// Mitsubishi GX Works2 project: PLC_Group_16   PLC: FX3G

// global labels: Global1
VAR_GLOBAL
  StartWorkingDay AT X010 : BOOL;
  In_Flour AT D1101 : REAL;
  Flour_Stock AT D1111 : REAL;
  check AT M0 : BOOL;
  In_Yeast AT D1103 : REAL;
  In_Water AT D1105 : REAL;
  In_Oil AT D1107 : REAL;
  In_Spice AT D1109 : REAL;
  Yeast_Stock AT D1113 : REAL;
  Water_Stock AT D1115 : REAL;
  Oil_Stock AT D1117 : REAL;
  Spice_Stock AT D1119 : REAL;
  Emergency_Button AT X007 : BOOL;
  Emg_Stop AT X007 : BOOL;
END_VAR
VAR_GLOBAL CONSTANT
  ratio1 : REAL := 0.2;
  Ratio_Yeast : REAL := 0.2;
END_VAR
VAR_GLOBAL
  Check_Yeast AT D1121 : REAL;
END_VAR
VAR_GLOBAL CONSTANT
  Ratio_Water : REAL := 0.5;
  Ratio_Oil : REAL := 0.3;
  Ratio_Spice : REAL := 0.1;
END_VAR
VAR_GLOBAL
  Check_Water AT D1123 : REAL;
  Check_Oil AT D1125 : REAL;
  Check_Spice AT D1127 : REAL;
END_VAR
VAR_GLOBAL CONSTANT
  MIN_Flour : REAL := 100.0;
END_VAR
VAR_GLOBAL
  checkY AT M1 : BOOL;
  checkW AT M2 : BOOL;
  checkO AT M3 : BOOL;
  checkS AT M4 : BOOL;
  checkF AT M5 : BOOL;
  active_workday AT Y010 : BOOL;
  M_10 AT M10 : BOOL;
  Start_Lisha AT X001 : BOOL;
  TC_1 AT TC1 : BOOL;
  TS_1 AT TS1 : BOOL;
  Lisha_Light AT Y001 : BOOL;
END_VAR
VAR_GLOBAL CONSTANT
  cons30 : INT := 30;
END_VAR
VAR_GLOBAL
  Water_Mixer AT D1131 : REAL;
  Flour_Mixer AT D1129 : REAL;
  Oil_Mixer AT D1133 : REAL;
  Spice_Mixer AT D1135 : REAL;
  Yeast_Mixer AT D1137 : REAL;
  Flour_Hatpaja AT D1139 : REAL;
  Water_Hatpaja AT D1141 : REAL;
  Yeat_Hatpaja AT D1143 : REAL;
  Oil_Hatpaja AT D1145 : REAL;
  Spice_Hatpaja AT D1147 : REAL;
  Flour_Bake AT D1149 : REAL;
  Water_Bake AT D1151 : REAL;
  Yeast_Bake AT D1153 : REAL;
  Oil_Bake AT D1155 : REAL;
  Spice_Bake AT D1157 : REAL;
  Flour_Store AT D1159 : REAL;
  Water_Store AT D1161 : REAL;
  Yeast_Store AT D1163 : REAL;
  Oil_Store AT D1165 : REAL;
  Spice_Store AT D1167 : REAL;
END_VAR
VAR_GLOBAL CONSTANT
  FlourCONS : REAL := 100;
  YeastCONS : REAL := 20;
  WaterCONS : REAL := 50;
  OilCONS : REAL := 30;
  SpiceCONS : REAL := 10;
END_VAR
VAR_GLOBAL
  checkREGISTER AT D1199 : REAL;
  Flour_Mehal AT D1169 : REAL;
  Water_Mehal AT D1171 : REAL;
  Oil_Mehal AT D1173 : REAL;
  Spice_Mehal AT D1175 : REAL;
  Yeast_Mehal AT D1177 : REAL;
  M_MEHAL AT M12 : BOOL;
  Start_Mehal AT X002 : BOOL;
  CC_1 AT CC1 : BOOL;
END_VAR
VAR_GLOBAL CONSTANT
  cons2 : INT := 2;
END_VAR
VAR_GLOBAL
  Start_Hatpaja AT X011 : BOOL;
  CS_1 AT CS1 : BOOL;
  Hachana_Light AT Y005 : BOOL;
  M_15 AT M15 : BOOL;
  M_11 AT M11 : BOOL;
  TC_2 AT TC2 : BOOL;
  TS_2 AT TS2 : BOOL;
  Hatpaja_Light_1 AT Y002 : BOOL;
  TC_3 AT TC3 : BOOL;
  TS_3 AT TS3 : BOOL;
  Hatpaja_Light_2 AT Y003 : BOOL;
END_VAR
VAR_GLOBAL CONSTANT
  cons20 : INT := 20;
END_VAR
VAR_GLOBAL
  TC_4 AT TC4 : BOOL;
END_VAR
VAR_GLOBAL CONSTANT
  Timer_3Sec : INT := 30;
END_VAR
VAR_GLOBAL
  TS_5 AT TS5 : BOOL;
  M_14 AT M14 : BOOL;
  TS_4 AT TS4 : BOOL;
END_VAR
VAR_GLOBAL CONSTANT
  cons5 : INT := 5;
END_VAR
VAR_GLOBAL
  TC_6 AT TC6 : BOOL;
END_VAR
VAR_GLOBAL CONSTANT
  cons40 : INT := 40;
END_VAR
VAR_GLOBAL
  TS_6 AT TS6 : BOOL;
  Bake_Light AT Y004 : BOOL;
  Start_Test AT X003 : BOOL;
  Analog_Input2 AT D8281 : INT;
  Analog_Test AT D8201 : INT;
END_VAR
VAR_GLOBAL CONSTANT
  Analog_Max : INT := 2000;
  Analog_Min : INT := 400;
END_VAR
VAR_GLOBAL
  M_6 AT M6 : BOOL;
  M_7 AT M7 : BOOL;
  TC_7 AT TC7 : BOOL;
  TS_7 AT TS7 : BOOL;
  Store_Light AT Y006 : BOOL;
  CC_3 AT CC3 : BOOL;
  CS_3 AT CS3 : BOOL;
  M_8 AT M8 : BOOL;
  TC_8 AT TC8 : BOOL;
  TC_9 AT TC9 : BOOL;
  TS_9 AT TS9 : BOOL;
  TC_10 AT TC10 : BOOL;
  M_30 AT M30 : BOOL;
  M_31 AT M31 : BOOL;
  TS_10 AT TS10 : BOOL;
END_VAR
VAR_GLOBAL CONSTANT
  Materials : BOOL := TRUE;
  Empty : BOOL;
END_VAR
VAR_GLOBAL
  M_32 AT M32 : BOOL;
  M_33 AT M33 : BOOL;
  FinishWorkingDay AT M34 : BOOL;
  M_40 AT M40 : BOOL;
  M_41 AT M41 : BOOL;
  M_42 AT M42 : BOOL;
  M_43 AT M43 : BOOL;
  M_44 AT M44 : BOOL;
  M_45 AT M45 : BOOL;
  M_46 AT M46 : BOOL;
  M_47 AT M47 : BOOL;
  M_48 AT M48 : BOOL;
  M_49 AT M49 : BOOL;
  M_FinishRound AT M50 : BOOL;
END_VAR
VAR_GLOBAL CONSTANT
  const0 : REAL;
END_VAR
VAR_GLOBAL
  M_88 AT M88 : BOOL;
  M_89 AT M89 : BOOL;
  M_90 AT M90 : BOOL;
  M_91 AT M91 : BOOL;
  M_92 AT M92 : BOOL;
  Ipus AT M99 : BOOL;
END_VAR
VAR_GLOBAL CONSTANT
  cons0 : REAL;
END_VAR
VAR_GLOBAL
  M_111 AT M111 : BOOL;
END_VAR

// task Task_01 (event TRUE, interval 0, priority 31): POU_01

PROGRAM POU_01
(* structured ladder/FBD written out as ST: instructions are called as NAME(EN, inputs, outputs); _pN, _eN, _tN stand for wires *)
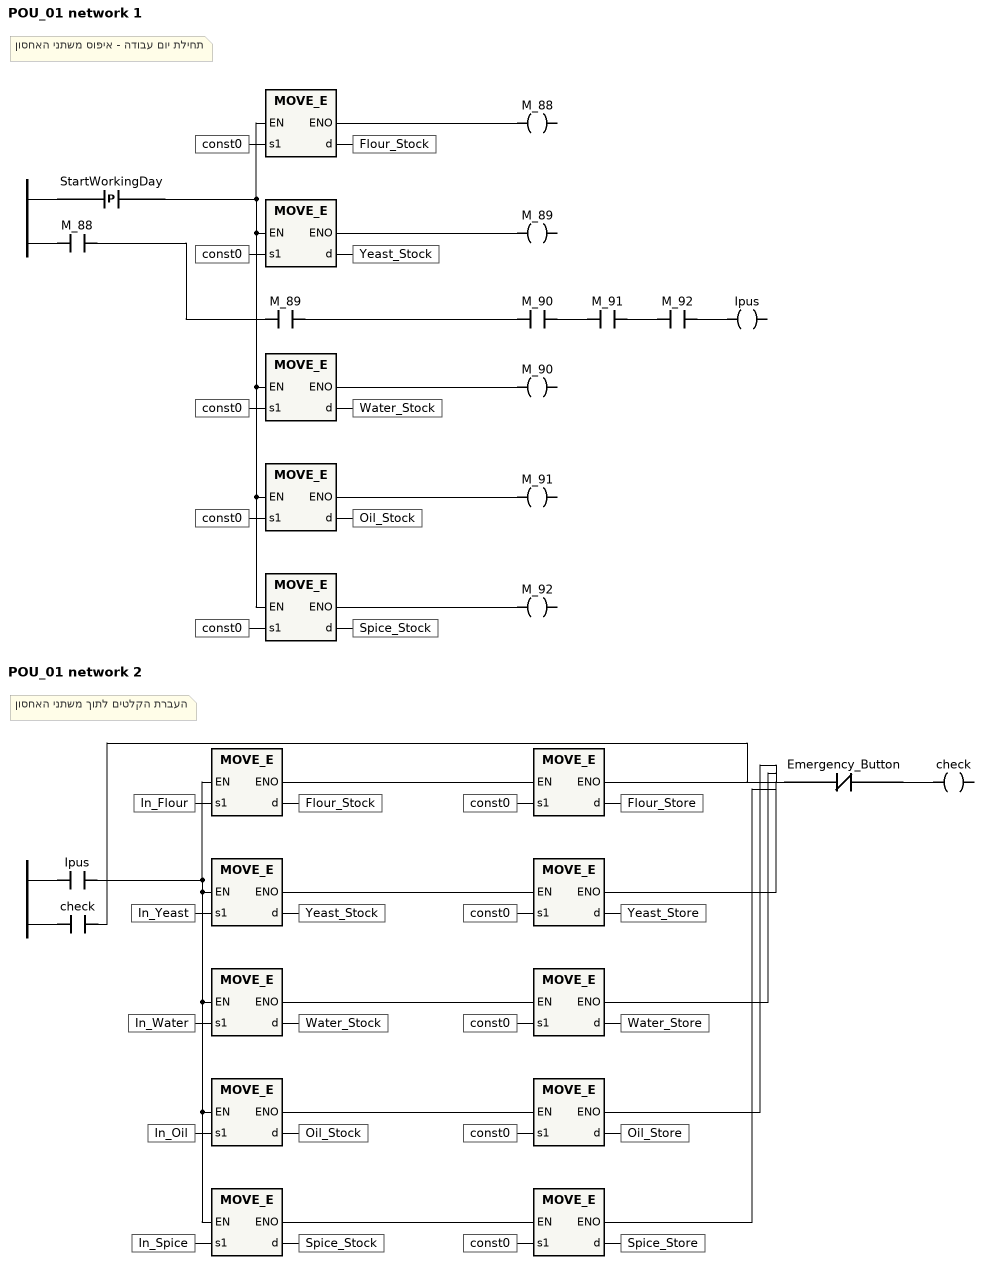
(* network 1 *)
(* תחילת יום עבודה - איפוס משתני האחסון *)
_p1 := LDP(TRUE, StartWorkingDay);
_e2 := MOVE_E(_p1, const0, Flour_Stock);
M_88 := _e2;
_e3 := MOVE_E(_p1, const0, Yeast_Stock);
M_89 := _e3;
_e4 := MOVE_E(_p1, const0, Water_Stock);
M_90 := _e4;
_e5 := MOVE_E(_p1, const0, Oil_Stock);
M_91 := _e5;
_e6 := MOVE_E(_p1, const0, Spice_Stock);
M_92 := _e6;
Ipus := M_88 AND M_89 AND M_90 AND M_91 AND M_92;
(* network 2 *)
(* העברת הקלטים לתוך משתני האחסון *)
_e1 := MOVE_E(Ipus, In_Flour, Flour_Stock);
_e2 := MOVE_E(_e1, const0, Flour_Store);
_e3 := MOVE_E(Ipus, In_Yeast, Yeast_Stock);
_e4 := MOVE_E(_e3, const0, Yeast_Store);
_e5 := MOVE_E(Ipus, In_Water, Water_Stock);
_e6 := MOVE_E(_e5, const0, Water_Store);
_e7 := MOVE_E(Ipus, In_Oil, Oil_Stock);
_e8 := MOVE_E(_e7, const0, Oil_Store);
_e9 := MOVE_E(Ipus, In_Spice, Spice_Stock);
_e10 := MOVE_E(_e9, const0, Spice_Store);
check := (_e2 OR _e4 OR _e6 OR _e8 OR _e10 OR check) AND NOT Emergency_Button;
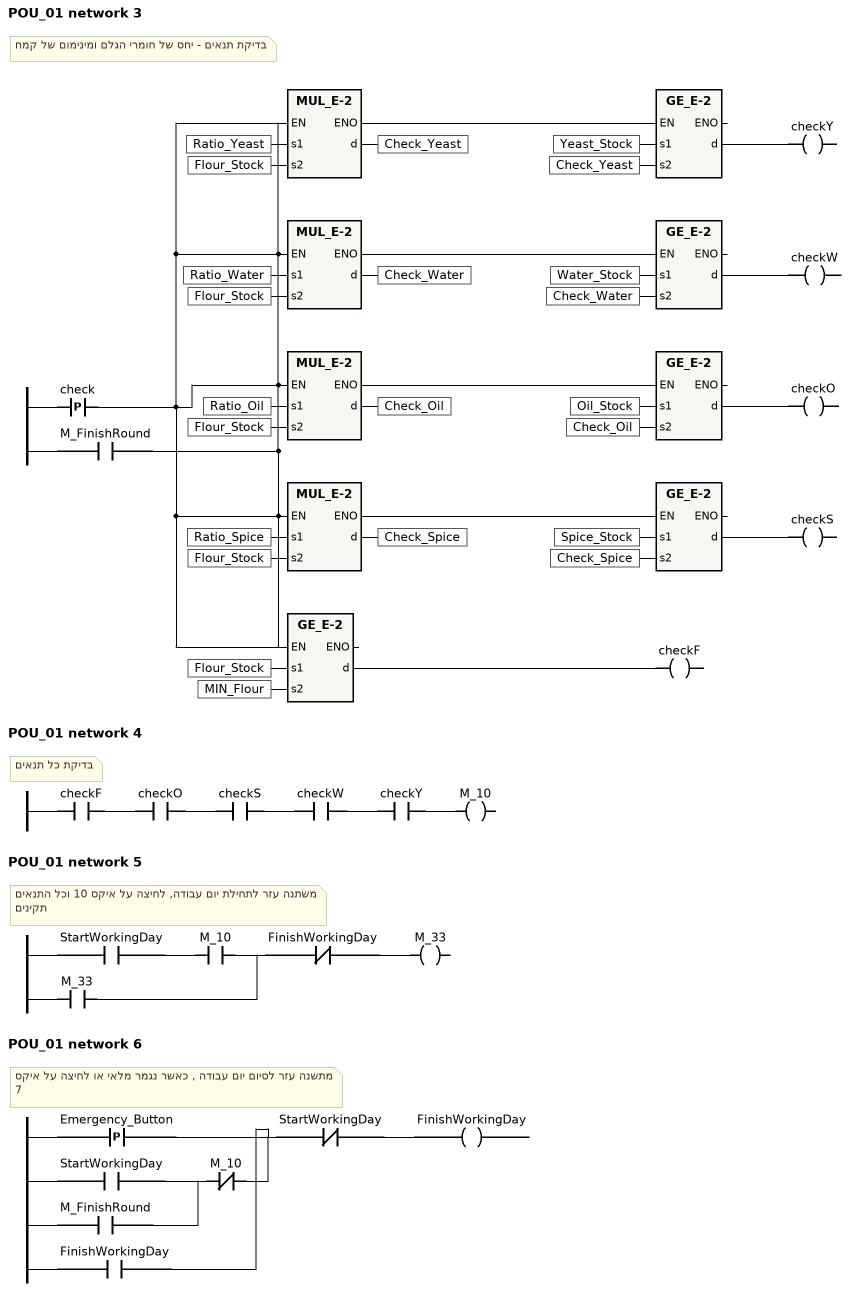
(* network 3 *)
(* בדיקת תנאים - יחס של חומרי הגלם ומינימום של קמח *)
_p1 := LDP(TRUE, check) OR M_FinishRound;
_e2 := MUL_E(_p1, Ratio_Yeast, Flour_Stock, Check_Yeast);
GE_E(_e2, Yeast_Stock, Check_Yeast, _t3);
checkY := _t3;
_e4 := MUL_E(_p1, Ratio_Water, Flour_Stock, Check_Water);
GE_E(_e4, Water_Stock, Check_Water, _t5);
checkW := _t5;
_e6 := MUL_E(_p1, Ratio_Oil, Flour_Stock, Check_Oil);
GE_E(_e6, Oil_Stock, Check_Oil, _t7);
checkO := _t7;
_e8 := MUL_E(_p1, Ratio_Spice, Flour_Stock, Check_Spice);
GE_E(_e8, Spice_Stock, Check_Spice, _t9);
checkS := _t9;
GE_E(_p1, Flour_Stock, MIN_Flour, _t10);
checkF := _t10;
(* network 4 *)
(* בדיקת כל תנאים *)
M_10 := checkF AND checkO AND checkS AND checkW AND checkY;
(* network 5 *)
(* משתנה עזר לתחילת יום עבודה, לחיצה על איקס 10 וכל התנאים תקינים *)
M_33 := ((StartWorkingDay AND M_10) OR M_33) AND NOT FinishWorkingDay;
(* network 6 *)
(* מתשנה עזר לסיום יום עבודה , כאשר נגמר מלאי או לחיצה על איקס 7 *)
FinishWorkingDay := (LDP(TRUE, Emergency_Button) OR ((StartWorkingDay OR M_FinishRound) AND NOT M_10) OR FinishWorkingDay) AND NOT StartWorkingDay;
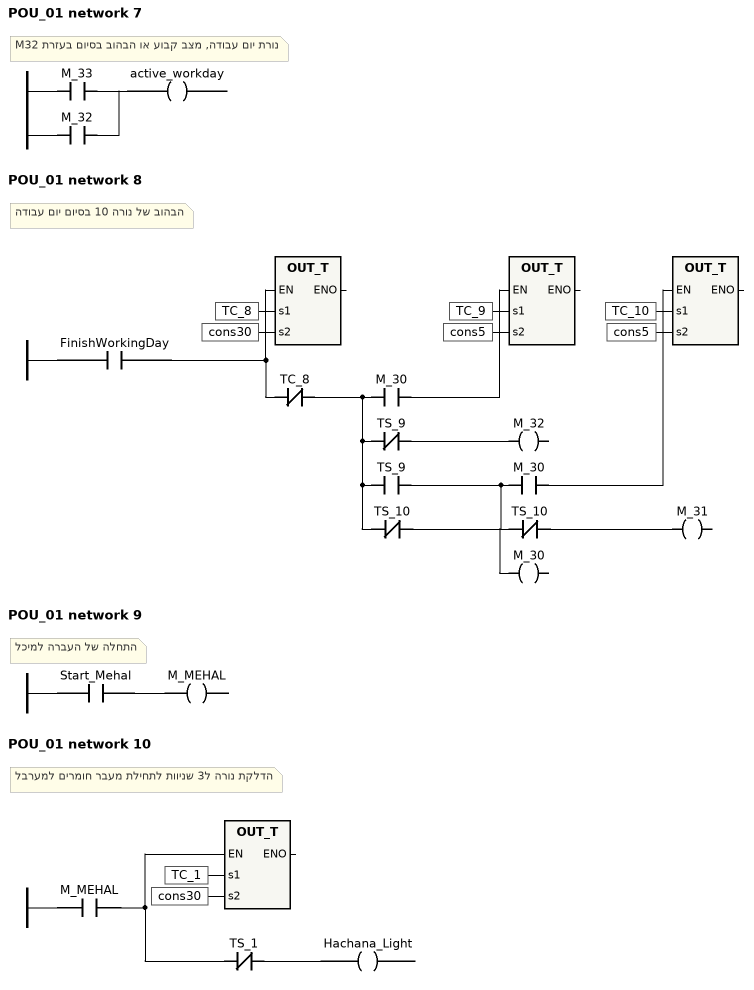
(* network 7 *)
(* נורת יום עבודה, מצב קבוע או הבהוב בסיום בעזרת M32 *)
active_workday := M_33 OR M_32;
(* network 8 *)
(* הבהוב של נורה 10 בסיום יום עבודה *)
OUT_T(FinishWorkingDay, TC_8, cons30);
_p1 := FinishWorkingDay AND NOT TC_8;
OUT_T(_p1 AND M_30, TC_9, cons5);
M_32 := _p1 AND NOT TS_9;
_p2 := _p1 AND TS_9;
OUT_T(_p2 AND M_30, TC_10, cons5);
M_31 := _p2 AND NOT TS_10;
M_30 := _p1 AND NOT TS_10;
(* network 9 *)
(* התחלה של העברה למיכל *)
M_MEHAL := Start_Mehal;
(* network 10 *)
(* הדלקת נורה ל3 שניוות לתחילת מעבר חומרים למערבל *)
OUT_T(M_MEHAL, TC_1, cons30);
Hachana_Light := M_MEHAL AND NOT TS_1;
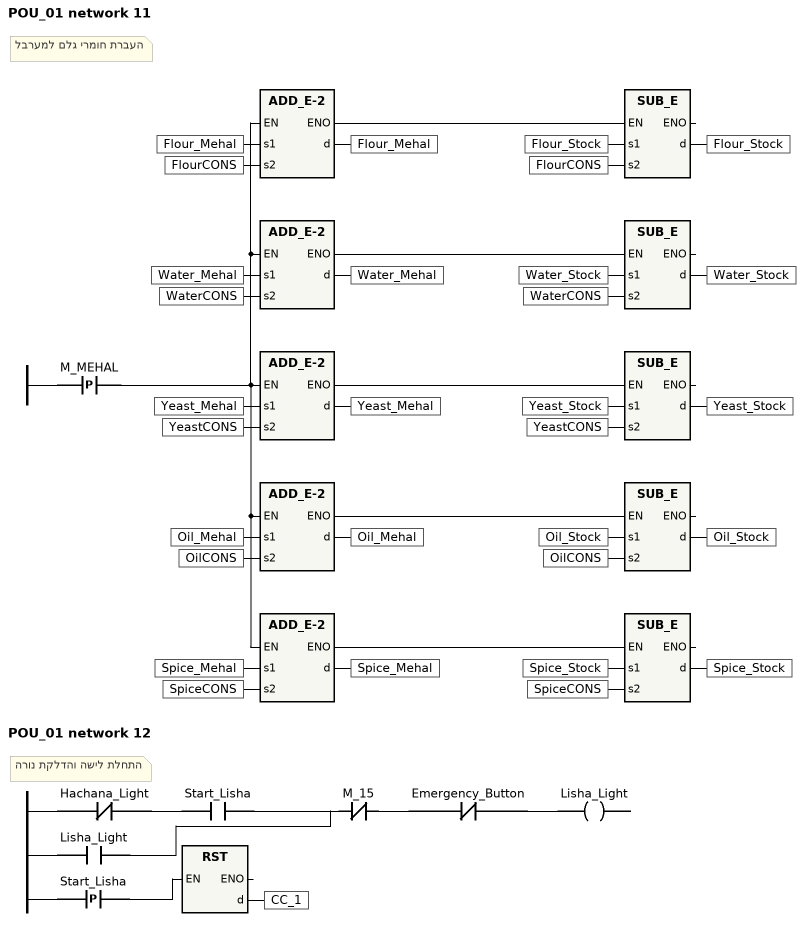
(* network 11 *)
(* העברת חומרי גלם למערבל *)
_p1 := LDP(TRUE, M_MEHAL);
_e2 := ADD_E(_p1, Flour_Mehal, FlourCONS, Flour_Mehal);
SUB_E(_e2, Flour_Stock, FlourCONS, Flour_Stock);
_e3 := ADD_E(_p1, Water_Mehal, WaterCONS, Water_Mehal);
SUB_E(_e3, Water_Stock, WaterCONS, Water_Stock);
_e4 := ADD_E(_p1, Yeast_Mehal, YeastCONS, Yeast_Mehal);
SUB_E(_e4, Yeast_Stock, YeastCONS, Yeast_Stock);
_e5 := ADD_E(_p1, Oil_Mehal, OilCONS, Oil_Mehal);
SUB_E(_e5, Oil_Stock, OilCONS, Oil_Stock);
_e6 := ADD_E(_p1, Spice_Mehal, SpiceCONS, Spice_Mehal);
SUB_E(_e6, Spice_Stock, SpiceCONS, Spice_Stock);
(* network 12 *)
(* התחלת לישה והדלקת נורה *)
Lisha_Light := (((NOT Hachana_Light AND Start_Lisha) OR Lisha_Light) AND NOT M_15) AND NOT Emergency_Button;
RST(LDP(TRUE, Start_Lisha), CC_1);
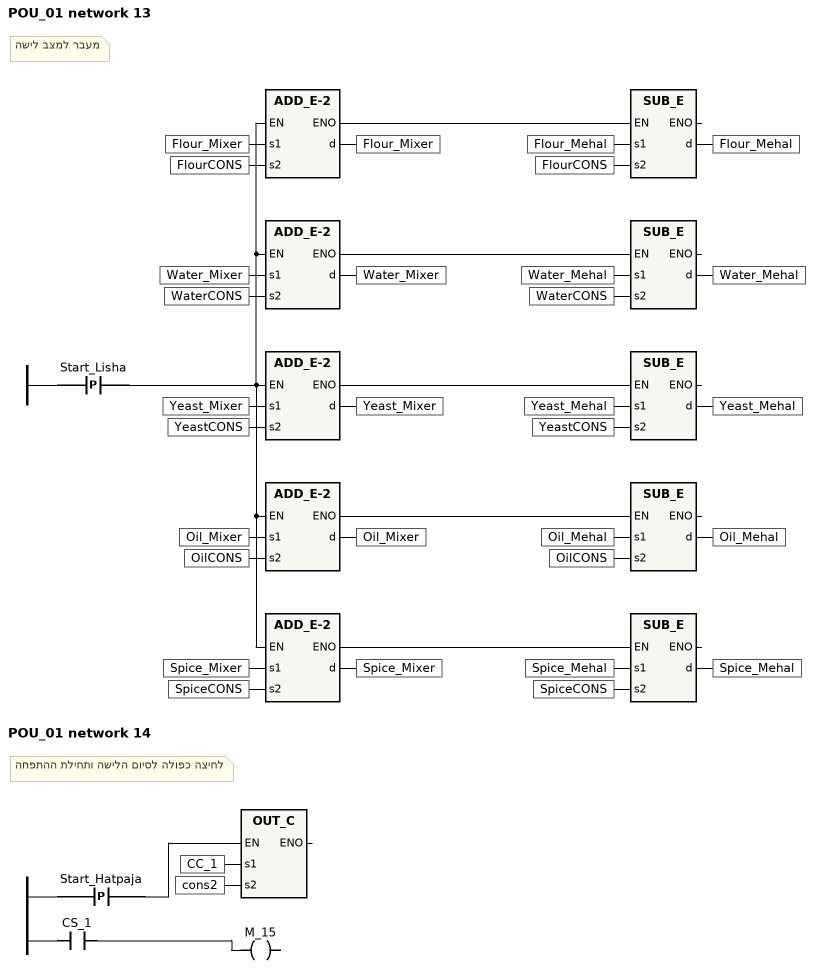
(* network 13 *)
(* מעבר למצב לישה *)
_p1 := LDP(TRUE, Start_Lisha);
_e2 := ADD_E(_p1, Flour_Mixer, FlourCONS, Flour_Mixer);
SUB_E(_e2, Flour_Mehal, FlourCONS, Flour_Mehal);
_e3 := ADD_E(_p1, Water_Mixer, WaterCONS, Water_Mixer);
SUB_E(_e3, Water_Mehal, WaterCONS, Water_Mehal);
_e4 := ADD_E(_p1, Yeast_Mixer, YeastCONS, Yeast_Mixer);
SUB_E(_e4, Yeast_Mehal, YeastCONS, Yeast_Mehal);
_e5 := ADD_E(_p1, Oil_Mixer, OilCONS, Oil_Mixer);
SUB_E(_e5, Oil_Mehal, OilCONS, Oil_Mehal);
_e6 := ADD_E(_p1, Spice_Mixer, SpiceCONS, Spice_Mixer);
SUB_E(_e6, Spice_Mehal, SpiceCONS, Spice_Mehal);
(* network 14 *)
(* לחיצה כפולה לסיום הלישה ותחילת ההתפחה *)
OUT_C(LDP(TRUE, Start_Hatpaja), CC_1, cons2);
M_15 := CS_1;
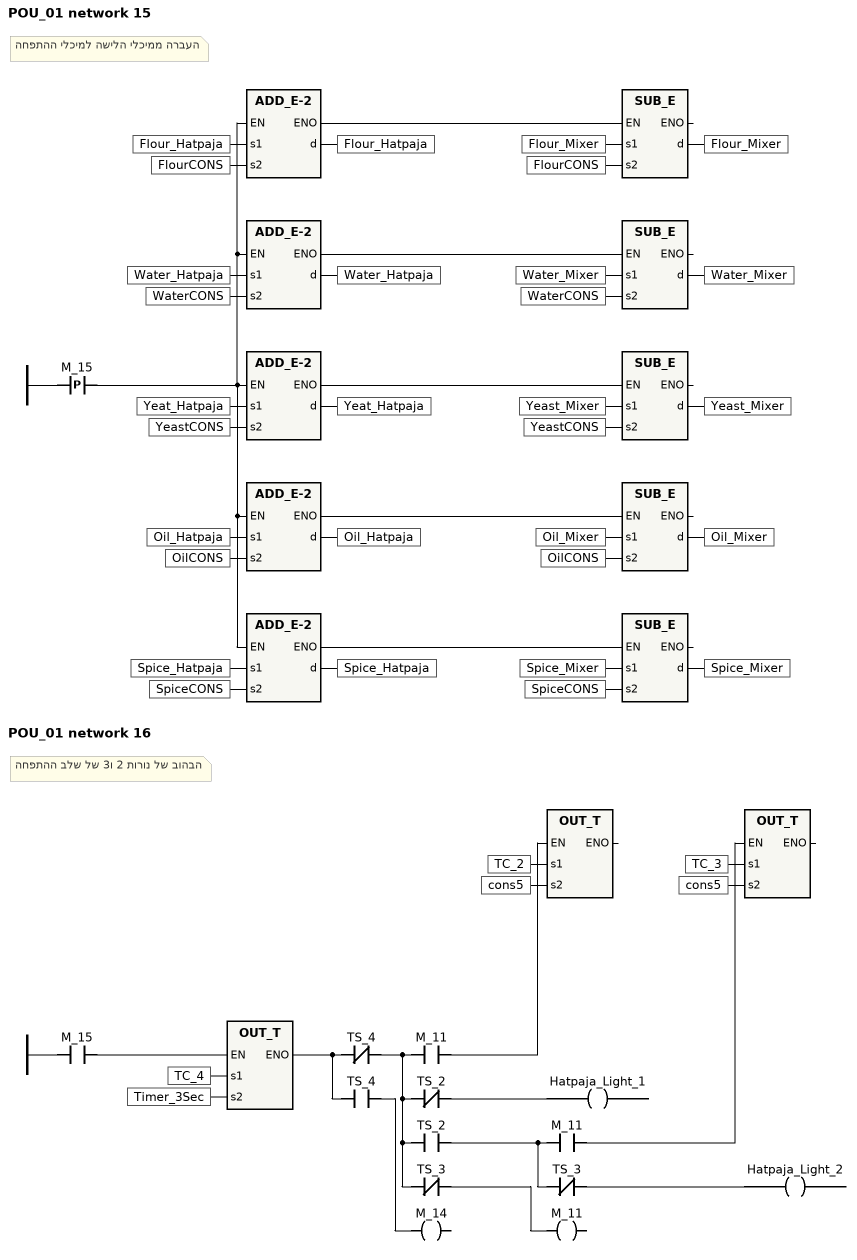
(* network 15 *)
(* העברה ממיכלי הלישה למיכלי ההתפחה *)
_p1 := LDP(TRUE, M_15);
_e2 := ADD_E(_p1, Flour_Hatpaja, FlourCONS, Flour_Hatpaja);
SUB_E(_e2, Flour_Mixer, FlourCONS, Flour_Mixer);
_e3 := ADD_E(_p1, Water_Hatpaja, WaterCONS, Water_Hatpaja);
SUB_E(_e3, Water_Mixer, WaterCONS, Water_Mixer);
_e4 := ADD_E(_p1, Yeat_Hatpaja, YeastCONS, Yeat_Hatpaja);
SUB_E(_e4, Yeast_Mixer, YeastCONS, Yeast_Mixer);
_e5 := ADD_E(_p1, Oil_Hatpaja, OilCONS, Oil_Hatpaja);
SUB_E(_e5, Oil_Mixer, OilCONS, Oil_Mixer);
_e6 := ADD_E(_p1, Spice_Hatpaja, SpiceCONS, Spice_Hatpaja);
SUB_E(_e6, Spice_Mixer, SpiceCONS, Spice_Mixer);
(* network 16 *)
(* הבהוב של נורות 2 ו3 של שלב ההתפחה *)
_e1 := OUT_T(M_15, TC_4, Timer_3Sec);
_p2 := _e1 AND NOT TS_4;
OUT_T(_p2 AND M_11, TC_2, cons5);
Hatpaja_Light_1 := _p2 AND NOT TS_2;
_p3 := _p2 AND TS_2;
OUT_T(_p3 AND M_11, TC_3, cons5);
Hatpaja_Light_2 := _p3 AND NOT TS_3;
M_11 := _p2 AND NOT TS_3;
M_14 := _e1 AND TS_4;
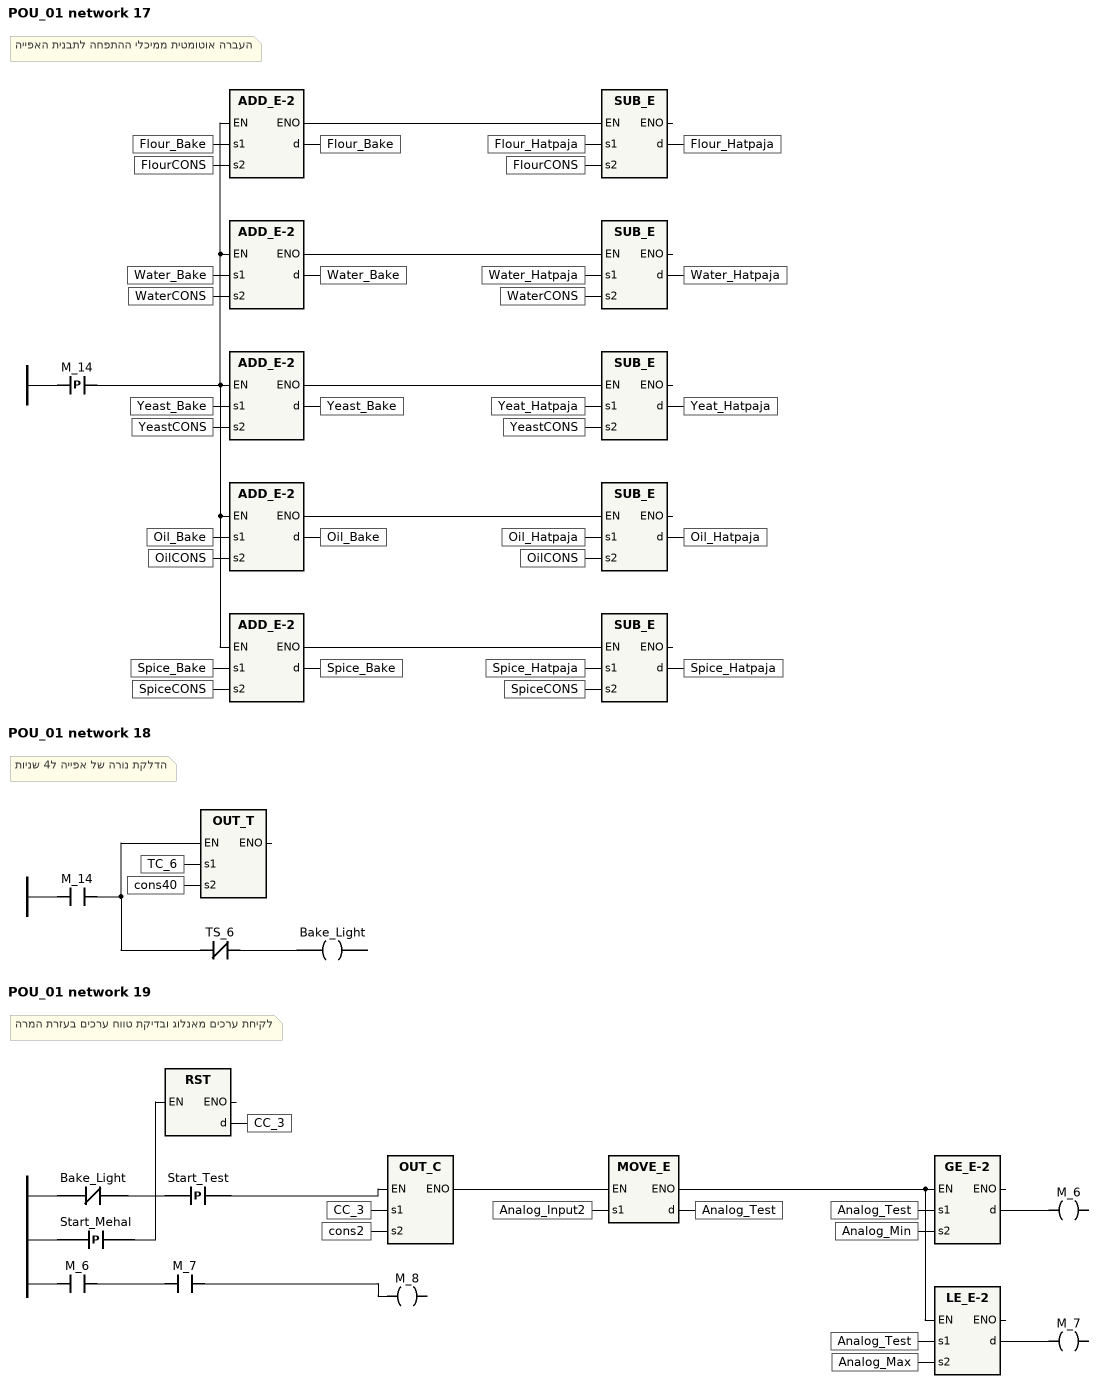
(* network 17 *)
(* העברה אוטומטית ממיכלי ההתפחה לתבנית האפייה *)
_p1 := LDP(TRUE, M_14);
_e2 := ADD_E(_p1, Flour_Bake, FlourCONS, Flour_Bake);
SUB_E(_e2, Flour_Hatpaja, FlourCONS, Flour_Hatpaja);
_e3 := ADD_E(_p1, Water_Bake, WaterCONS, Water_Bake);
SUB_E(_e3, Water_Hatpaja, WaterCONS, Water_Hatpaja);
_e4 := ADD_E(_p1, Yeast_Bake, YeastCONS, Yeast_Bake);
SUB_E(_e4, Yeat_Hatpaja, YeastCONS, Yeat_Hatpaja);
_e5 := ADD_E(_p1, Oil_Bake, OilCONS, Oil_Bake);
SUB_E(_e5, Oil_Hatpaja, OilCONS, Oil_Hatpaja);
_e6 := ADD_E(_p1, Spice_Bake, SpiceCONS, Spice_Bake);
SUB_E(_e6, Spice_Hatpaja, SpiceCONS, Spice_Hatpaja);
(* network 18 *)
(* הדלקת נורה של אפייה ל4 שניות *)
OUT_T(M_14, TC_6, cons40);
Bake_Light := M_14 AND NOT TS_6;
(* network 19 *)
(* לקיחת ערכים מאנלוג ובדיקת טווח ערכים בעזרת המרה *)
_e1 := OUT_C(NOT Bake_Light AND LDP(TRUE, Start_Test), CC_3, cons2);
_e2 := MOVE_E(_e1, Analog_Input2, Analog_Test);
GE_E(_e2, Analog_Test, Analog_Min, _t3);
M_6 := _t3;
RST(LDP(TRUE, Start_Mehal), CC_3);
LE_E(_e2, Analog_Test, Analog_Max, _t4);
M_7 := _t4;
M_8 := M_6 AND M_7;
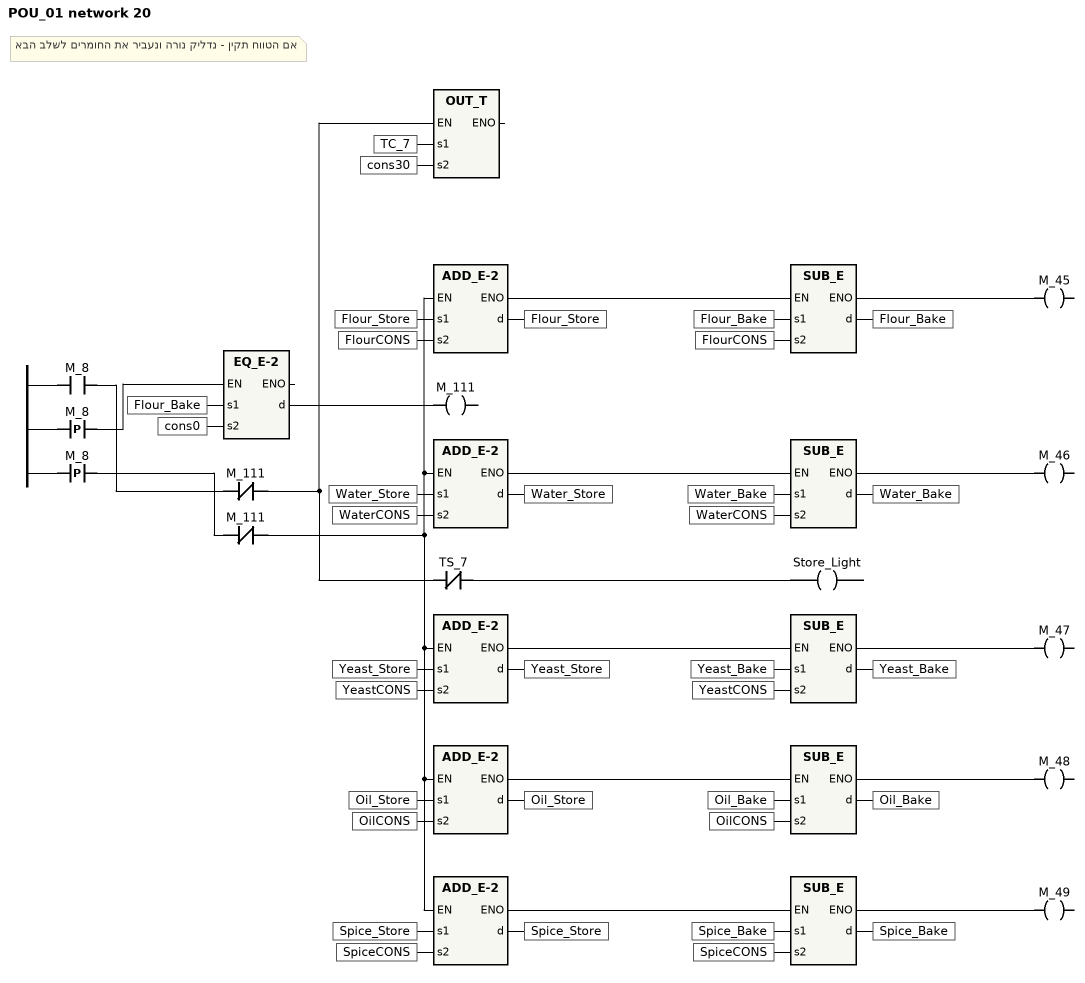
(* network 20 *)
(* אם הטווח תקין - נדליק נורה ונעביר את החומרים לשלב הבא *)
_p1 := M_8 AND NOT M_111;
OUT_T(_p1, TC_7, cons30);
Store_Light := _p1 AND NOT TS_7;
EQ_E(LDP(TRUE, M_8), Flour_Bake, cons0, _t2);
M_111 := _t2;
_p3 := LDP(TRUE, M_8) AND NOT M_111;
_e4 := ADD_E(_p3, Flour_Store, FlourCONS, Flour_Store);
_e5 := SUB_E(_e4, Flour_Bake, FlourCONS, Flour_Bake);
M_45 := _e5;
_e6 := ADD_E(_p3, Water_Store, WaterCONS, Water_Store);
_e7 := SUB_E(_e6, Water_Bake, WaterCONS, Water_Bake);
M_46 := _e7;
_e8 := ADD_E(_p3, Yeast_Store, YeastCONS, Yeast_Store);
_e9 := SUB_E(_e8, Yeast_Bake, YeastCONS, Yeast_Bake);
M_47 := _e9;
_e10 := ADD_E(_p3, Oil_Store, OilCONS, Oil_Store);
_e11 := SUB_E(_e10, Oil_Bake, OilCONS, Oil_Bake);
M_48 := _e11;
_e12 := ADD_E(_p3, Spice_Store, SpiceCONS, Spice_Store);
_e13 := SUB_E(_e12, Spice_Bake, SpiceCONS, Spice_Bake);
M_49 := _e13;
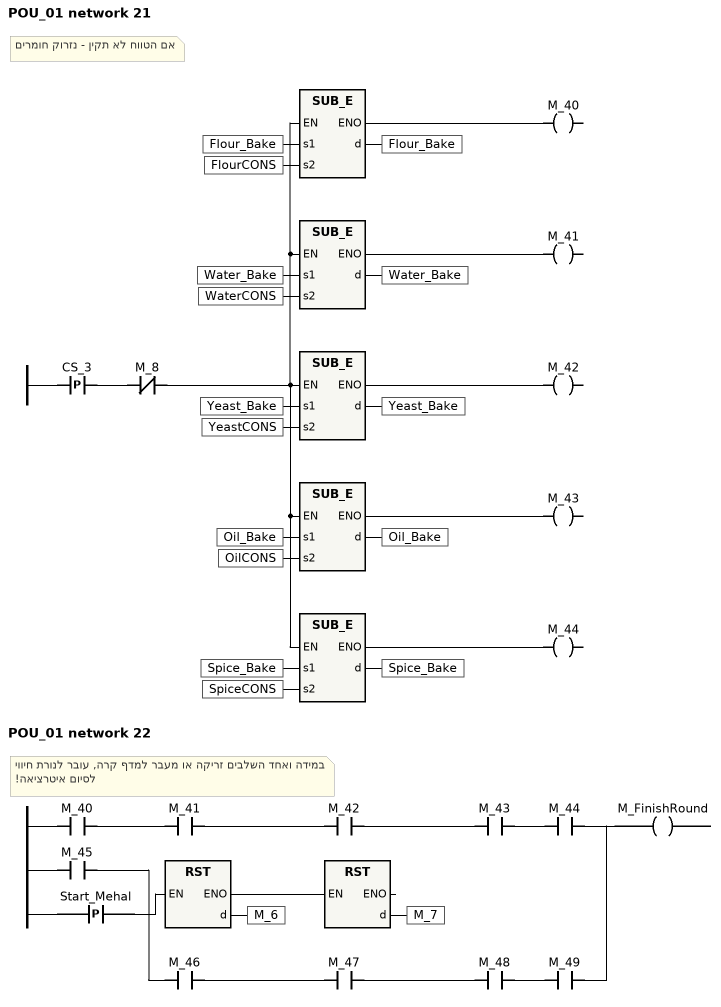
(* network 21 *)
(* אם הטווח לא תקין - נזרוק חומרים *)
_p1 := LDP(TRUE, CS_3) AND NOT M_8;
_e2 := SUB_E(_p1, Flour_Bake, FlourCONS, Flour_Bake);
M_40 := _e2;
_e3 := SUB_E(_p1, Water_Bake, WaterCONS, Water_Bake);
M_41 := _e3;
_e4 := SUB_E(_p1, Yeast_Bake, YeastCONS, Yeast_Bake);
M_42 := _e4;
_e5 := SUB_E(_p1, Oil_Bake, OilCONS, Oil_Bake);
M_43 := _e5;
_e6 := SUB_E(_p1, Spice_Bake, SpiceCONS, Spice_Bake);
M_44 := _e6;
(* network 22 *)
(* במידה ואחד השלבים זריקה או מעבר למדף קרה, עובר לנורת חיווי  לסיום איטרציאה! *)
M_FinishRound := (M_40 AND M_41 AND M_42 AND M_43 AND M_44) OR (M_45 AND M_46 AND M_47 AND M_48 AND M_49);
_e1 := RST(LDP(TRUE, Start_Mehal), M_6);
RST(_e1, M_7);
END_PROGRAM
